# EPICS autosave request: stdApp/Db/throttle.req
$(P)$(THR).PREC
$(P)$(THR).DPREC
$(P)$(THR).OUT
$(P)$(THR).DLY
$(P)$(THR).VAL
$(P)$(THR).DRVLC
$(P)$(THR).DRVLL
$(P)$(THR).DRVLH
$(P)$(THR).SINP
